(* IEC 61131-3 sources: pcworx-testkit/export-st, 4 files *)

(* ---- Concole.IEC ---- *)
(*@PROPERTIES_EX@
TYPE: DATA_TYPE
LOCALE: 0
*)
TYPE
	ARR_STR_0_1000 : ARRAY [0 ..1000] OF STRING;

	udtConsole	:
	STRUCT
		iCounter: INT;
		arrData: ARR_STR_0_1000;
	END_STRUCT;
END_TYPE

(* ---- IL_RS_UNI.IEC ---- *)
(*@PROPERTIES_EX@
TYPE: DATA_TYPE
LOCALE: 0
*)
TYPE

	ARR_B_0_13 : ARRAY [0..13] OF BYTE;

	udtRS485Frame	:
	STRUCT
		iCounter	:	INT;
		iWordsNo	:	INT;
		arrData		:	ARR_B_0_13;
	END_STRUCT;

	udtBufferReceive :
	STRUCT
		iWordsNo 	: INT;
		arrData		: ARR_B_0_13;
	END_STRUCT;

	udtBufferSend :
	STRUCT
		iWordsNo 	: INT;
		arrData		: ARR_B_0_13;
	END_STRUCT;
END_TYPE

(* ---- Console.ST ---- *)
(*@PROPERTIES_EX@
TYPE: POU
LOCALE: 0
IEC_LANGUAGE: ST
PLC_TYPE: independent
PROC_TYPE: independent
GROUP: Debug
*)
(*@KEY@:DESCRIPTION*)

(*@KEY@:END_DESCRIPTION*)
FUNCTION_BLOCK Console

(*Group:Default*)

VAR_EXTERNAL
	PLC_SYS_TICK_CNT :	DINT;(*Number of system ticks*)
END_VAR

VAR
	strDelimeter :	STRING;
END_VAR

VAR_INPUT
	strSource :	STRING;
	strMessage :	STRING;
END_VAR

VAR_EXTERNAL
	udtConsole :	udtConsole;
END_VAR

VAR
	strConsole :	STRING;
	iConsoleCounter :	INT;
END_VAR

(*@KEY@: WORKSHEET
NAME: Console
IEC_LANGUAGE: ST
*)
strDelimeter						:= ';';

strConsole							:= DINT_TO_STRING(PLC_SYS_TICK_CNT, '%d');
strConsole							:= CONCAT(strConsole, strDelimeter);

strConsole							:= CONCAT(strConsole, strSource);
strConsole							:= CONCAT(strConsole, strDelimeter);

strConsole							:= CONCAT(strConsole, strMessage);

IF udtConsole.iCounter >= 1000
THEN
	iConsoleCounter					:= 0;
ELSE
	iConsoleCounter					:= udtConsole.iCounter + 1;
END_IF;

udtConsole.arrData[iConsoleCounter] := strConsole;
udtConsole.iCounter					:= iConsoleCounter;
(*@KEY@: END_WORKSHEET *)
END_FUNCTION_BLOCK

(* ---- IL_UNI07.ST ---- *)
(*@PROPERTIES_EX@
TYPE: POU
LOCALE: 0
IEC_LANGUAGE: ST
PLC_TYPE: independent
PROC_TYPE: independent
GROUP: Serial
*)
(*@KEY@:DESCRIPTION*)

(*@KEY@:END_DESCRIPTION*)
FUNCTION_BLOCK IL_UNI07

(*Group:Inputs*)

VAR_INPUT
	xConsoleLog :	BOOL;
	strConsoleId :	STRING;
END_VAR

(*Group:Inouts*)

VAR_IN_OUT
	udtRS485Line :	udtRS485Frame;
	arrInputAddress :	MB2_RSUNI_ARR_B_1_14;(*Process Data Input*)
	arrOutputAddress :	MB2_RSUNI_ARR_B_1_14;(*Process Data Output*)
END_VAR

(*Group:FB*)

VAR
	R_TRIG_xSending :	R_TRIG;
	Console :	Console;
END_VAR

(*Group:Internal*)

VAR
	udtBufferReceive :	udtBufferReceive;
	udtBufferSend :	udtBufferSend;
	xSending :	BOOL;
	iByteNum :	INT;
	iBytesToCopy :	INT;
	bStatusBits :	BYTE;
	wNumberOfCharactersReceived :	WORD;
	iFirstAddressIndex :	INT;
	iLastAddressIndex :	INT;
	iAddressIndex :	INT;
	iFirstBufferIndex :	INT;
	iByteToCopy :	INT;
	iWordsTransmitted :	INT;
	iWordsReceived :	INT;
	wWordsReceived :	WORD;
	wWordsTransmitted :	WORD;
	udtRS485Line_iCounterPrev :	INT;
	iWordsToSend :	INT;
END_VAR

(*@KEY@: WORKSHEET
NAME: IL_UNI07
IEC_LANGUAGE: ST
*)
(* ========================================== Clearing data ===================================================== *)
FOR iByteToCopy	:= 1 TO 14 DO

	arrOutputAddress[iByteToCopy] := BYTE#16#00;

END_FOR;
(* ============================================================================================================== *)

(* ============================================= Module status bits ============================================= *)
bStatusBits.X0 := udtBufferReceive.iWordsNo > 0; 	(* Receive buffer not empty *)
bStatusBits.X1 := FALSE; 							(* Receive error *)
bStatusBits.X2 := FALSE; 							(* Transmit error *)
bStatusBits.X3 := FALSE; 							(* DCD *)
bStatusBits.X4 := FALSE; 							(* Receive buffer full *)
bStatusBits.X5 := FALSE; 							(* Transmit buffer full*)
bStatusBits.X6 := udtBufferSend.iWordsNo > 0; 		(* Transmit buffer not empty *)
bStatusBits.X7 := FALSE;							(* DSR *)

(* =============================================================================================================== *)

(* ======================================== Execute commands ======================================================*)

(* "Read number of characters received" command *)
IF arrInputAddress[1] = BYTE#16#00 THEN

	IF xConsoleLog THEN
		Console.strSource				:= strConsoleId;
		Console.strMessage				:= CONCAT('ReadNumberOfChar command, number ', INT_TO_STRING(udtBufferReceive.iWordsNo, '%d'));
		Console();
	END_IF;

	arrOutputAddress[1] 			:= arrInputAddress[1];						(* Command mirror *)
	arrOutputAddress[2] 			:= bStatusBits;								(* Status bits *)

	wNumberOfCharactersReceived 	:= INT_TO_WORD(udtBufferReceive.iWordsNo);
	arrOutputAddress[3] 			:= wNumberOfCharactersReceived.B0;
	arrOutputAddress[4] 			:= wNumberOfCharactersReceived.B1;

(* “Transmit characters” command *)
ELSIF arrInputAddress[1] = BYTE#16#10
	OR arrInputAddress[1] = BYTE#16#50
	AND NOT xSending
	THEN

		IF xConsoleLog THEN
			Console.strSource			:= strConsoleId;
			Console.strMessage			:= 'TransmitChar command';
			Console();
		END_IF;

		iWordsToSend				:= BYTE_TO_INT(arrInputAddress[3]);
		iBytesToCopy				:= iWordsToSend * 2;

		arrOutputAddress[1] 		:= arrInputAddress[1];						(* Command mirror *)
		arrOutputAddress[2] 		:= bStatusBits;								(* Status bits *)

		iFirstAddressIndex			:= 4;
		iLastAddressIndex			:= MIN(iBytesToCopy - 1, 14);
		iFirstBufferIndex			:= 0;

		FOR iAddressIndex := iFirstAddressIndex TO iLastAddressIndex DO
			udtBufferSend.arrData[iFirstBufferIndex] 	:= arrInputAddress[iAddressIndex];
			iFirstBufferIndex 							:= iFirstBufferIndex + 1;
		END_FOR;

		udtBufferSend.iWordsNo		:= iWordsToSend;

		xSending					:= TRUE;

(* "Read characters" command *)
ELSIF arrInputAddress[1] = BYTE#16#30 THEN

	IF xConsoleLog THEN
		Console.strSource			:= strConsoleId;
		Console.strMessage			:= CONCAT('ReadChar command, length ', INT_TO_STRING(udtBufferReceive.iWordsNo, '%d'));
		Console();
	END_IF;

	arrOutputAddress[1] 		:= arrInputAddress[1];						(* Command mirror *)
	bStatusBits.X0 				:= FALSE;
	arrOutputAddress[2] 		:= bStatusBits;								(* Status bits *)

	arrOutputAddress[3] 		:= INT_TO_BYTE(udtBufferReceive.iWordsNo);	(* Number of valid characters available in the input data *)

	iBytesToCopy 				:= udtBufferReceive.iWordsNo * 2;

	iFirstAddressIndex			:= 4;
	iLastAddressIndex			:= MIN(iFirstAddressIndex + iBytesToCopy - 1, 14);
	iFirstBufferIndex			:= 0;
	FOR iAddressIndex := iFirstAddressIndex TO iLastAddressIndex DO
		arrOutputAddress[iAddressIndex] := udtBufferReceive.arrData[iFirstBufferIndex];
		iFirstBufferIndex 				:= iFirstBufferIndex + 1;
	END_FOR;

	udtBufferReceive.iWordsNo	:= 0;

(* "Read counters" command *)
ELSIF arrInputAddress[1] = BYTE#16#3E
	AND arrInputAddress[2] = BYTE#16#00 THEN

		IF xConsoleLog THEN
			Console.strSource			:= strConsoleId;
			Console.strMessage			:= 'ReadCounters command';
			Console();
		END_IF;

		arrOutputAddress[1] 		:= arrInputAddress[1];						(* Command mirror *)
		arrOutputAddress[2] 		:= bStatusBits;								(* Status bits *)

		wWordsReceived				:= INT_TO_WORD(iWordsReceived);
		arrOutputAddress[3]			:= wWordsReceived.B0;
		arrOutputAddress[4]			:= wWordsReceived.B1;

		wWordsTransmitted			:= INT_TO_WORD(iWordsTransmitted);
		arrOutputAddress[7]			:= wWordsTransmitted.B0;
		arrOutputAddress[8]			:= wWordsTransmitted.B1;

(* "Write configuration" command *)
ELSIF arrInputAddress[1] = BYTE#16#40 THEN

	IF xConsoleLog THEN
		Console.strSource			:= strConsoleId;
		Console.strMessage			:= 'Write configuration command';
		Console();
	END_IF;

	arrOutputAddress[1] 		:= arrInputAddress[1];						(* Command mirror *)
	arrOutputAddress[2] 		:= bStatusBits;								(* Status bits *)

ELSE

	IF xConsoleLog THEN
		Console.strSource			:= strConsoleId;
		Console.strMessage			:= CONCAT(BYTE_TO_STRING(arrInputAddress[1], '%x'),' command');
		Console();
	END_IF;

	arrOutputAddress[1] 		:= 	arrInputAddress[1];						(* Command mirror *)

END_IF;

(* ============================================================================================================== *)

(* ==================================== Clear xSending flag if command is changing ============================== *)
IF arrInputAddress[1] <> BYTE#16#10
	AND arrInputAddress[1] <> BYTE#16#50
	THEN

		xSending	:= FALSE;

END_IF;

R_TRIG_xSending.CLK	:= xSending;
R_TRIG_xSending();
(* ============================================================================================================== *)

(* ================================= Sending data from internal buffer to serial interface ====================== *)
IF R_TRIG_xSending.Q
	AND udtBufferSend.iWordsNo > 0 THEN

		IF xConsoleLog THEN
			Console.strSource			:= strConsoleId;
			Console.strMessage			:= CONCAT('Sending to interface, length ', INT_TO_STRING(udtBufferSend.iWordsNo, '%d'));
			Console();
		END_IF;

		iBytesToCopy :=  MIN((udtBufferSend.iWordsNo * 2) - 1, 13);

		FOR iByteNum := 0 TO iBytesToCopy DO

			udtRS485Line.arrData[iByteNum] := udtBufferSend.arrData[iByteNum];

		END_FOR;

		udtRS485Line.iCounter		:= udtRS485Line.iCounter + 1;
		udtRS485Line.iWordsNo		:= udtBufferSend.iWordsNo;
		udtRS485Line_iCounterPrev 	:= udtRS485Line.iCounter;

		udtBufferSend.iWordsNo		:= 0;

(* ======================================== Copy data from interface to internal buffer ======================= *)
ELSIF udtRS485Line.iCounter > udtRS485Line_iCounterPrev
	AND NOT xSending
	AND udtRS485Line.iWordsNo > 0 THEN

		IF xConsoleLog THEN
			Console.strSource				:= strConsoleId;
			Console.strMessage				:= CONCAT('Receiving from interface, length ', INT_TO_STRING(udtRS485Line.iWordsNo, '%d'));
			Console();
		END_IF;

		iBytesToCopy :=  MIN((udtRS485Line.iWordsNo * 2) - 1, 13);

		FOR iByteNum := 0 TO iBytesToCopy DO

			udtBufferReceive.arrData[iByteNum] := udtRS485Line.arrData[iByteNum];

		END_FOR;

		udtBufferReceive.iWordsNo	:= udtRS485Line.iWordsNo;
		iWordsReceived				:= iWordsReceived + udtRS485Line.iWordsNo;
		udtRS485Line_iCounterPrev 	:= udtRS485Line.iCounter;

END_IF;
(* ============================================================================================================== *)

(*@KEY@: END_WORKSHEET *)
END_FUNCTION_BLOCK
